PROGRAM POUNCPowerOn
VAR
	fbAxis1PowerOn:MC_Power;
	fbAxis2PowerOn:MC_Power;
	fbAxis3PowerOn:MC_Power;
	fbAxis4PowerOn:MC_Power;
	fbAxis5PowerOn:MC_Power;
	fbAxis6PowerOn:MC_Power;
	bAxis1LimitPosI AT%I* :BOOL;
	bAxis1LimitNegI AT%I* :BOOL;
	bAxis2LimitPosI AT%I* :BOOL;
	bAxis2LimitNegI AT%I* :BOOL;
	bAxis3LimitPosI AT%I* :BOOL;
	bAxis3LimitNegI AT%I* :BOOL;
	bAxis4LimitPosI AT%I* :BOOL;
	bAxis4LimitNegI AT%I* :BOOL;
	bAxis5LimitPosI AT%I* :BOOL;
	bAxis5LimitNegI AT%I* :BOOL;
	bAxis6LimitPosI AT%I* :BOOL;
	bAxis6LimitNegI AT%I* :BOOL;
END_VAR

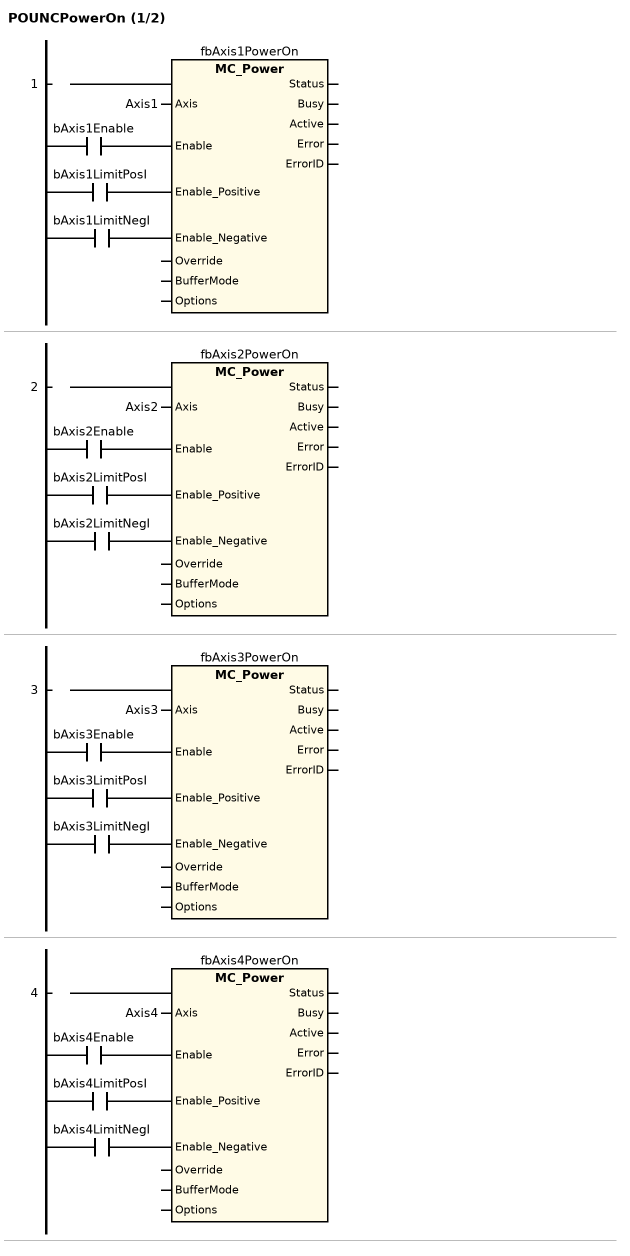
// NETWORK 1
fbAxis1PowerOn(
    Axis := Axis1,
    Enable := bAxis1Enable,
    Enable_Positive := bAxis1LimitPosI,
    Enable_Negative := bAxis1LimitNegI); // MC_Power

// NETWORK 2
fbAxis2PowerOn(
    Axis := Axis2,
    Enable := bAxis2Enable,
    Enable_Positive := bAxis2LimitPosI,
    Enable_Negative := bAxis2LimitNegI); // MC_Power

// NETWORK 3
fbAxis3PowerOn(
    Axis := Axis3,
    Enable := bAxis3Enable,
    Enable_Positive := bAxis3LimitPosI,
    Enable_Negative := bAxis3LimitNegI); // MC_Power

// NETWORK 4
fbAxis4PowerOn(
    Axis := Axis4,
    Enable := bAxis4Enable,
    Enable_Positive := bAxis4LimitPosI,
    Enable_Negative := bAxis4LimitNegI); // MC_Power

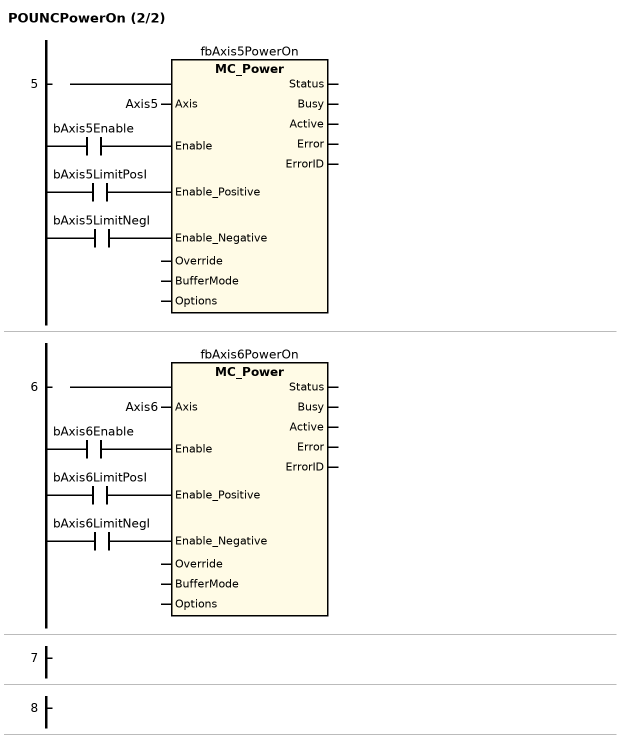
// NETWORK 5
fbAxis5PowerOn(
    Axis := Axis5,
    Enable := bAxis5Enable,
    Enable_Positive := bAxis5LimitPosI,
    Enable_Negative := bAxis5LimitNegI); // MC_Power

// NETWORK 6
fbAxis6PowerOn(
    Axis := Axis6,
    Enable := bAxis6Enable,
    Enable_Positive := bAxis6LimitPosI,
    Enable_Negative := bAxis6LimitNegI); // MC_Power

// NETWORK 7

// NETWORK 8

END_PROGRAM

(* stored: Version 1.1.0.1, ProductVersion 3.1.4022.18
   POU POUNCPowerOn: Id {10652921-91f0-48f4-8e4f-e05ddb809ef3}, SpecialFunc None *)
